{attribute addProperty BoxType "EPP6001-0002-0016"}
{attribute addProperty Id "StatusAT %I*UINT1621Data_InAT %I*ARRAY[0 ..21] OF USINT176220"}
{attribute addProperty CRC "2032034109"}
{attribute addProperty SizeInBites "192"}
{attribute addProperty SizeInBytes "24"}
TYPE COM_Inputs_18212A5E :
STRUCT
	{attribute addProperty Name "Status"}
	Status AT %I* : UINT;
	{attribute addProperty Name "Data_In"}
	Data_In AT %I* : ARRAY[0 ..21] OF USINT;
END_STRUCT
END_TYPE

(* stored: Version 1.2.0.0, ProductVersion 3.1.4024.9
   DUT COM_Inputs_18212A5E: Id {10395afe-7d11-4af5-95b5-94ed2215caa6} *)
